PROGRAM MAIN
VAR
	fbCycleTimeLogger	: FB_LogTaskCycleTime := (nCycleInterval:=1000);
END_VAR

IF _TaskInfo[1].FirstCycle THEN
	// Change AMS id if log service runs on different server than
	// plc. Remove if plc and service runs on the same machine.
	//PRG_TaskLog.Init('192.168.56.1.1.1');
	F_Log(E_LogLevel.eInfo, 'Plc started.');
END_IF

// simulates load on the task
PRG_SimulateLoad();

// simulate logs
PRG_SimulateLogs();

// logs the cycle time statistics
fbCycleTimeLogger();

PRG_TaskLog.Call();

END_PROGRAM

(* stored: Version 1.1.0.1, ProductVersion 3.1.4022.10
   POU MAIN: Id {21bfe353-a59a-4092-b9d6-97dae9bf59b4}, SpecialFunc None *)
